///Interface for barcode readers result subscriber
INTERFACE IBarcodeReaderSubscriber

// New data recieved
METHOD NewDataRecieved : HResult
VAR_INPUT
    data : Data; ///Data recieved
    result : BarcodeCodeReadingResult; ///Reading result
END_VAR
END_METHOD

END_INTERFACE

(* stored: Version 1.1.0.1, ProductVersion 3.1.4020.12
   Itf IBarcodeReaderSubscriber: Id {9f259c6a-4048-4115-bfa6-c75047605960}
   Method NewDataRecieved: Id {e457b818-c9ed-42ed-bc70-b22ec68a0536} *)
